(* Schneider Machine Expert - Basic project PLC_getstart, file version 1.8.0.0 *)
(* ProjectInformations: Name=New project *)

HARDWARE
  Cpu 0: TM221CE16R
  EthernetConfiguration: NetworkName=M221, IpAllocationMode=FixedAddress, IpAddress=0.0.0.0, SubnetMask=0.0.0.0
  SerialLineConfiguration: Baud=Baud19200, Parity=ParityEven, DataBits=DataBits8, StopBits=StopBits1, PhysicalMedium=PhysicalMediumRs485, TransmissionMode=TransmissionModeModbusRtu, SlaveId=1, Addressing=SlaveAddressing
  MastTask: UsePeriodScanMode=false, PeriodScan=100
  FastTask: Period=255
  CpuBehavior: StartingMode=StartAsPreviousState, AutoSaveRamOnEeprom=true, WatchdogPeriod=250

SYMBOLS  (address, symbol, comment, settings)
  %M0       MEM_SW_BLK
  %M1       MEM_RUN_H
  %M2       MEM_LRED
  %M3       MEM_LYLW
  %M4       MEM_LGRN
  %M5       MEM_RUN_L
  %M6       MEM_SW_GRN
  %TM0      DLY_YLW_BOFF  [Preset=7, Base=OneHundredMilliSeconds, IsRetentive=true]
  %TM1      DLY_YLW_ON  [Preset=10, Base=OneHundredMilliSeconds, IsRetentive=true]
  %TM2      DLY_RED_ON  [Preset=50, Base=OneHundredMilliSeconds, IsRetentive=true]
  %TM3      DLY_GRN_ON  [Preset=20, Base=OneHundredMilliSeconds, IsRetentive=true]
  %TM4      DLY_YLW_BON  [Preset=7, Base=OneHundredMilliSeconds, IsRetentive=true]
  %TM5      DLY_YLW_MON  [Preset=15, Base=OneHundredMilliSeconds, IsRetentive=true]
  %I0.0     SW_RED
  %I0.1     SW_BLK
  %I0.2     SW_GRN
  %Q0.0     LAMP_YLW
  %Q0.1     LAMP_GRN
  %Q0.2     LAMP_RED

POU Mode Select
  (* SectionNumber=1 *)

// Rung 0
  LD %M0                  (* MEM_SW_BLK *)
  ANDN %M1                (* MEM_RUN_H *)
  AND %M5                 (* MEM_RUN_L *)
  S %M1                   (* MEM_RUN_H *)
  S %M5                   (* MEM_RUN_L *)
  R %M0                   (* MEM_SW_BLK *)
  // as ST:
  //   _t1 := MEM_SW_BLK AND NOT MEM_RUN_H AND MEM_RUN_L;
  //   IF _t1 THEN MEM_RUN_H := TRUE; END_IF;
  //   IF _t1 THEN MEM_RUN_L := TRUE; END_IF;
  //   IF _t1 THEN MEM_SW_BLK := FALSE; END_IF;
  (* the ladder stored for this rung does not match its IL; not drawn *)

POU Process RGY
  (* SectionNumber=2 *)

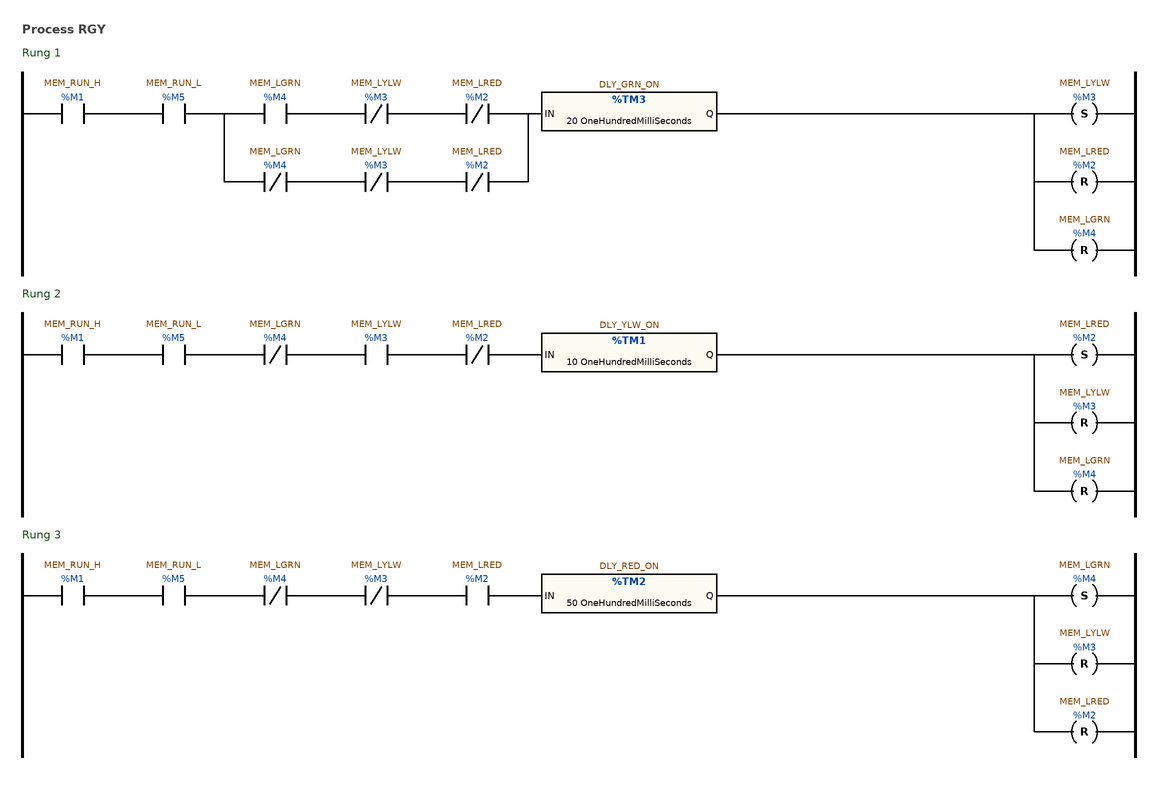

// Rung 1
  BLK %TM3                (* DLY_GRN_ON *)
  LD %M1                  (* MEM_RUN_H *)
  AND %M5                 (* MEM_RUN_L *)
  AND( %M4                (* MEM_LGRN *)
  ANDN %M3                (* MEM_LYLW *)
  ANDN %M2                (* MEM_LRED *)
  OR(N %M4                (* MEM_LGRN *)
  ANDN %M3                (* MEM_LYLW *)
  ANDN %M2                (* MEM_LRED *)
  )
  )
  IN
  OUT_BLK
  LD Q
  S %M3                   (* MEM_LYLW *)
  R %M2                   (* MEM_LRED *)
  R %M4                   (* MEM_LGRN *)
  END_BLK
  // as ST:
  //   DLY_GRN_ON(IN := MEM_RUN_H AND MEM_RUN_L AND (MEM_LGRN AND NOT MEM_LYLW AND NOT MEM_LRED OR NOT MEM_LGRN AND NOT MEM_LYLW AND NOT MEM_LRED));
  //   IF DLY_GRN_ON.Q THEN MEM_LYLW := TRUE; END_IF;
  //   IF DLY_GRN_ON.Q THEN MEM_LRED := FALSE; END_IF;
  //   IF DLY_GRN_ON.Q THEN MEM_LGRN := FALSE; END_IF;

// Rung 2
  BLK %TM1                (* DLY_YLW_ON *)
  LD %M1                  (* MEM_RUN_H *)
  AND %M5                 (* MEM_RUN_L *)
  ANDN %M4                (* MEM_LGRN *)
  AND %M3                 (* MEM_LYLW *)
  ANDN %M2                (* MEM_LRED *)
  IN
  OUT_BLK
  LD Q
  S %M2                   (* MEM_LRED *)
  R %M3                   (* MEM_LYLW *)
  R %M4                   (* MEM_LGRN *)
  END_BLK
  // as ST:
  //   DLY_YLW_ON(IN := MEM_RUN_H AND MEM_RUN_L AND NOT MEM_LGRN AND MEM_LYLW AND NOT MEM_LRED);
  //   IF DLY_YLW_ON.Q THEN MEM_LRED := TRUE; END_IF;
  //   IF DLY_YLW_ON.Q THEN MEM_LYLW := FALSE; END_IF;
  //   IF DLY_YLW_ON.Q THEN MEM_LGRN := FALSE; END_IF;

// Rung 3
  BLK %TM2                (* DLY_RED_ON *)
  LD %M1                  (* MEM_RUN_H *)
  AND %M5                 (* MEM_RUN_L *)
  ANDN %M4                (* MEM_LGRN *)
  ANDN %M3                (* MEM_LYLW *)
  AND %M2                 (* MEM_LRED *)
  IN
  OUT_BLK
  LD Q
  S %M4                   (* MEM_LGRN *)
  R %M3                   (* MEM_LYLW *)
  R %M2                   (* MEM_LRED *)
  END_BLK
  // as ST:
  //   DLY_RED_ON(IN := MEM_RUN_H AND MEM_RUN_L AND NOT MEM_LGRN AND NOT MEM_LYLW AND MEM_LRED);
  //   IF DLY_RED_ON.Q THEN MEM_LGRN := TRUE; END_IF;
  //   IF DLY_RED_ON.Q THEN MEM_LYLW := FALSE; END_IF;
  //   IF DLY_RED_ON.Q THEN MEM_LRED := FALSE; END_IF;

POU Process Ylw
  (* SectionNumber=3 *)

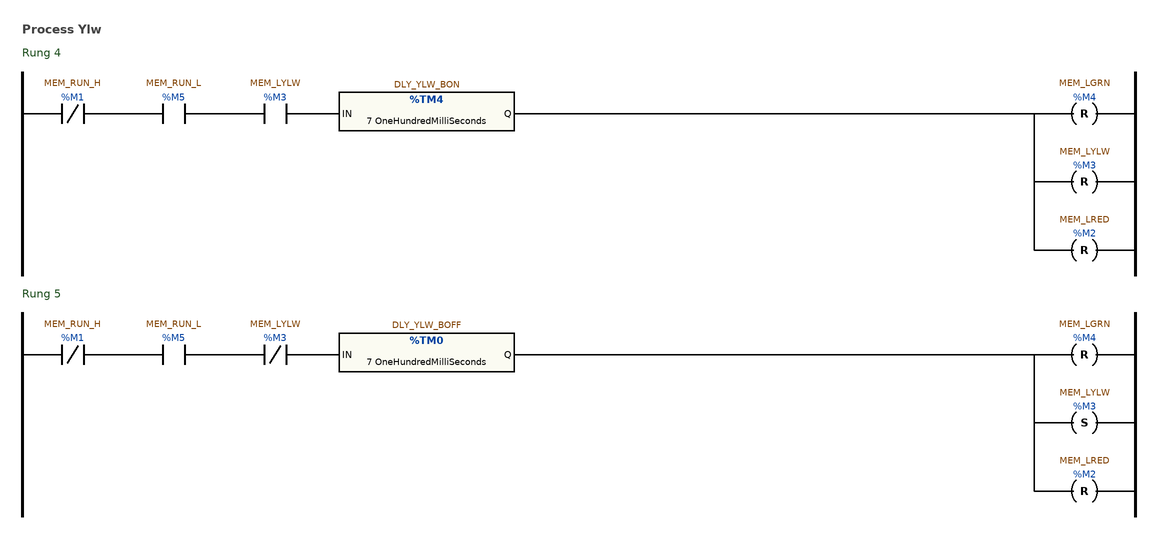

// Rung 4
  BLK %TM4                (* DLY_YLW_BON *)
  LDN %M1                 (* MEM_RUN_H *)
  AND %M5                 (* MEM_RUN_L *)
  AND %M3                 (* MEM_LYLW *)
  IN
  OUT_BLK
  LD Q
  R %M4                   (* MEM_LGRN *)
  R %M3                   (* MEM_LYLW *)
  R %M2                   (* MEM_LRED *)
  END_BLK
  // as ST:
  //   DLY_YLW_BON(IN := NOT MEM_RUN_H AND MEM_RUN_L AND MEM_LYLW);
  //   IF DLY_YLW_BON.Q THEN MEM_LGRN := FALSE; END_IF;
  //   IF DLY_YLW_BON.Q THEN MEM_LYLW := FALSE; END_IF;
  //   IF DLY_YLW_BON.Q THEN MEM_LRED := FALSE; END_IF;

// Rung 5
  BLK %TM0                (* DLY_YLW_BOFF *)
  LDN %M1                 (* MEM_RUN_H *)
  AND %M5                 (* MEM_RUN_L *)
  ANDN %M3                (* MEM_LYLW *)
  IN
  OUT_BLK
  LD Q
  R %M4                   (* MEM_LGRN *)
  S %M3                   (* MEM_LYLW *)
  R %M2                   (* MEM_LRED *)
  END_BLK
  // as ST:
  //   DLY_YLW_BOFF(IN := NOT MEM_RUN_H AND MEM_RUN_L AND NOT MEM_LYLW);
  //   IF DLY_YLW_BOFF.Q THEN MEM_LGRN := FALSE; END_IF;
  //   IF DLY_YLW_BOFF.Q THEN MEM_LYLW := TRUE; END_IF;
  //   IF DLY_YLW_BOFF.Q THEN MEM_LRED := FALSE; END_IF;

POU Process Manual
  (* SectionNumber=4 *)

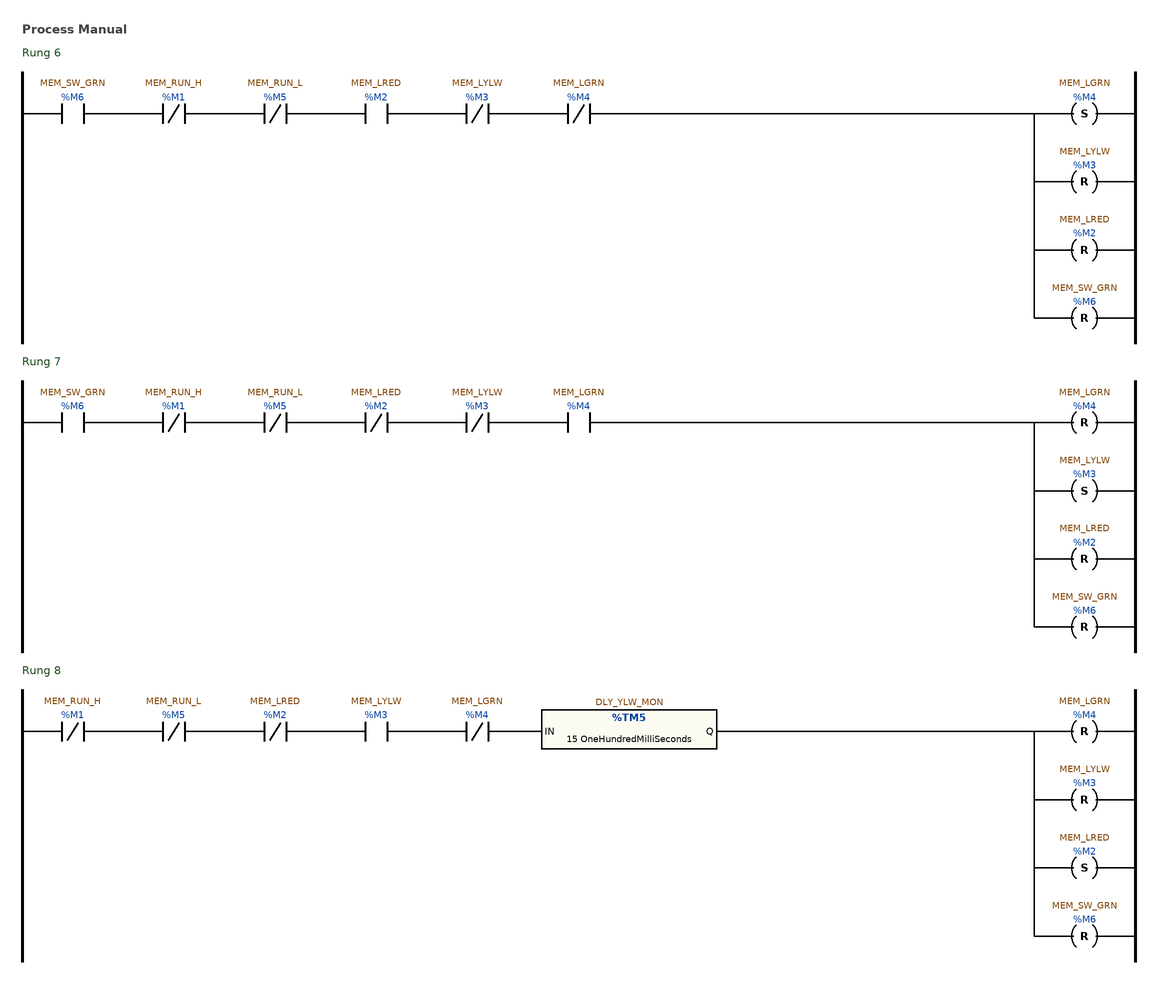

// Rung 6
  LD %M6                  (* MEM_SW_GRN *)
  ANDN %M1                (* MEM_RUN_H *)
  ANDN %M5                (* MEM_RUN_L *)
  AND %M2                 (* MEM_LRED *)
  ANDN %M3                (* MEM_LYLW *)
  ANDN %M4                (* MEM_LGRN *)
  S %M4                   (* MEM_LGRN *)
  R %M3                   (* MEM_LYLW *)
  R %M2                   (* MEM_LRED *)
  R %M6                   (* MEM_SW_GRN *)
  // as ST:
  //   _t1 := MEM_SW_GRN AND NOT MEM_RUN_H AND NOT MEM_RUN_L AND MEM_LRED AND NOT MEM_LYLW AND NOT MEM_LGRN;
  //   IF _t1 THEN MEM_LGRN := TRUE; END_IF;
  //   IF _t1 THEN MEM_LYLW := FALSE; END_IF;
  //   IF _t1 THEN MEM_LRED := FALSE; END_IF;
  //   IF _t1 THEN MEM_SW_GRN := FALSE; END_IF;

// Rung 7
  LD %M6                  (* MEM_SW_GRN *)
  ANDN %M1                (* MEM_RUN_H *)
  ANDN %M5                (* MEM_RUN_L *)
  ANDN %M2                (* MEM_LRED *)
  ANDN %M3                (* MEM_LYLW *)
  AND %M4                 (* MEM_LGRN *)
  R %M4                   (* MEM_LGRN *)
  S %M3                   (* MEM_LYLW *)
  R %M2                   (* MEM_LRED *)
  R %M6                   (* MEM_SW_GRN *)
  // as ST:
  //   _t1 := MEM_SW_GRN AND NOT MEM_RUN_H AND NOT MEM_RUN_L AND NOT MEM_LRED AND NOT MEM_LYLW AND MEM_LGRN;
  //   IF _t1 THEN MEM_LGRN := FALSE; END_IF;
  //   IF _t1 THEN MEM_LYLW := TRUE; END_IF;
  //   IF _t1 THEN MEM_LRED := FALSE; END_IF;
  //   IF _t1 THEN MEM_SW_GRN := FALSE; END_IF;

// Rung 8
  BLK %TM5                (* DLY_YLW_MON *)
  LDN %M1                 (* MEM_RUN_H *)
  ANDN %M5                (* MEM_RUN_L *)
  ANDN %M2                (* MEM_LRED *)
  AND %M3                 (* MEM_LYLW *)
  ANDN %M4                (* MEM_LGRN *)
  IN
  OUT_BLK
  LD Q
  R %M4                   (* MEM_LGRN *)
  R %M3                   (* MEM_LYLW *)
  S %M2                   (* MEM_LRED *)
  R %M6                   (* MEM_SW_GRN *)
  END_BLK
  // as ST:
  //   DLY_YLW_MON(IN := NOT MEM_RUN_H AND NOT MEM_RUN_L AND NOT MEM_LRED AND MEM_LYLW AND NOT MEM_LGRN);
  //   IF DLY_YLW_MON.Q THEN MEM_LGRN := FALSE; END_IF;
  //   IF DLY_YLW_MON.Q THEN MEM_LYLW := FALSE; END_IF;
  //   IF DLY_YLW_MON.Q THEN MEM_LRED := TRUE; END_IF;
  //   IF DLY_YLW_MON.Q THEN MEM_SW_GRN := FALSE; END_IF;

POU MAP IO
  (* SectionNumber=5 *)

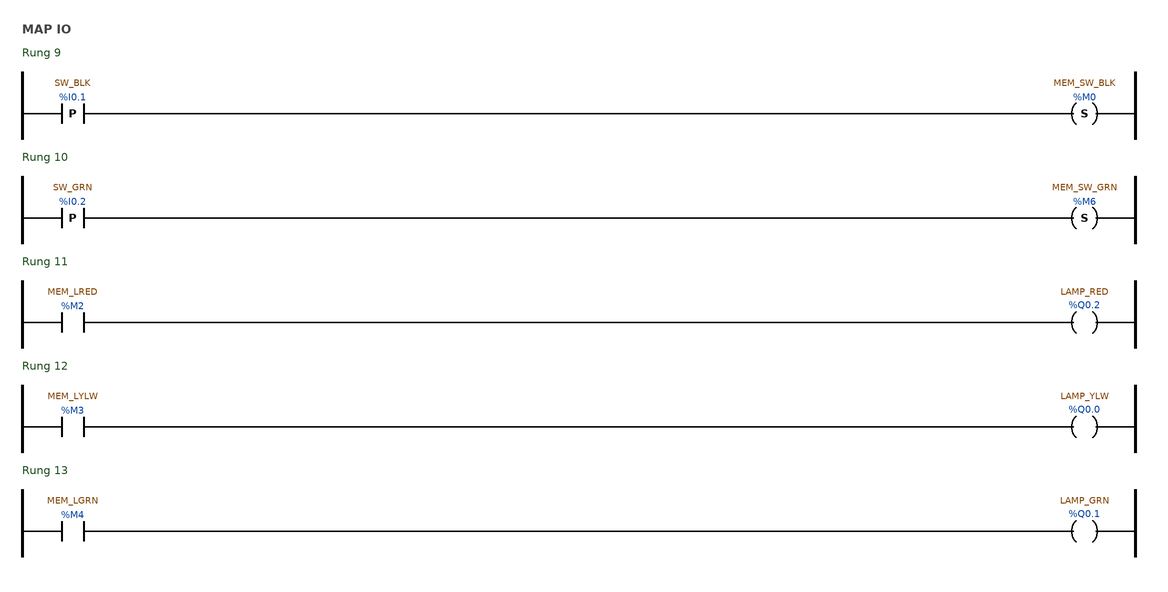

// Rung 9
  LDR %I0.1               (* SW_BLK *)
  S %M0                   (* MEM_SW_BLK *)
  // as ST:
  //   IF RISING(SW_BLK) THEN MEM_SW_BLK := TRUE; END_IF;

// Rung 10
  LDR %I0.2               (* SW_GRN *)
  S %M6                   (* MEM_SW_GRN *)
  // as ST:
  //   IF RISING(SW_GRN) THEN MEM_SW_GRN := TRUE; END_IF;

// Rung 11
  LD %M2                  (* MEM_LRED *)
  ST %Q0.2                (* LAMP_RED *)
  // as ST:
  //   LAMP_RED := MEM_LRED;

// Rung 12
  LD %M3                  (* MEM_LYLW *)
  ST %Q0.0                (* LAMP_YLW *)
  // as ST:
  //   LAMP_YLW := MEM_LYLW;

// Rung 13
  LD %M4                  (* MEM_LGRN *)
  ST %Q0.1                (* LAMP_GRN *)
  // as ST:
  //   LAMP_GRN := MEM_LGRN;
